Fanuc KAREL source: kf00088.KL

-- PROVISIONAL review KL for V770-1; original PC SHA256 11a14ad524d03e6830a47306cda54a4af466bb7a67b4344e7b336353ae99738e
-- Incomplete behavior may be omitted. Consult companion uncertainty JSON. Do not deploy.
PROGRAM KF00088
%NOLOCKGROUP
BEGIN
  -- UNRESOLVED_PC offsets 5-28; opcodes 27,22,1C,31,4A
  -- UNRESOLVED_PC offsets 33-37; opcodes 7F
END KF00088
